FUNCTION_BLOCK TLController (* Composite Function Block Type *)
  (* Standard: 61499-2 *)
  (* Version 0.2, 2003-12-05, JHC, Rockwell Automation, Renamed from NEWCOMPFB. *)
  (* Version 0.1, 2002-01-08, JHC, Rockwell Automation, Added DLY FB as example. *)
  (* Version 0.0, 2000-05-27, JHC, Rockwell Automation *)
  (* Compiler header: package fb.rt.template; *)
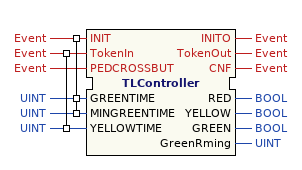
  EVENT_INPUT
    INIT WITH GREENTIME, MINGREENTIME; (* Initialization Request *)
    TokenIn WITH YELLOWTIME;
    PEDCROSSBUT;
  END_EVENT
  EVENT_OUTPUT
    INITO; (* Initialization Confirm *)
    TokenOut;
    CNF;
  END_EVENT
  VAR_INPUT
    GREENTIME : UINT;
    MINGREENTIME : UINT;
    YELLOWTIME : UINT;
  END_VAR
  VAR_OUTPUT
    RED : BOOL;
    YELLOW : BOOL;
    GREEN : BOOL;
    GreenRming : UINT;
  END_VAR
  FBS
    ButPressCTR : E_CTU(PV := 4);
    CLOCK : E_CYCLE(DT := t#1s);
    Split1 : E_SPLIT;
    Controller1 : Controller;
  END_FBS
  EVENT_CONNECTIONS
    PEDCROSSBUT TO ButPressCTR.CU;
    Split1.EO1 TO TokenOut;
    Split1.EO2 TO CLOCK.STOP;
    INIT TO CLOCK.START;
    TokenIn TO CLOCK.START;
    INIT TO Controller1.INIT;
    CLOCK.EO TO Controller1.CLK;
    TokenIn TO Controller1.LD;
    Controller1.INITO TO INITO;
    Controller1.CNF TO CNF;
  END_CONNECTIONS
  DATA_CONNECTIONS
    Controller1.RED TO RED;
    Controller1.YELLOW TO YELLOW;
    Controller1.GREEN TO GREEN;
    Controller1.GREENREMAINING TO GreenRming;
    ButPressCTR.Q TO Controller1.PEDCROSS;
    GREENTIME TO Controller1.GREENTIME;
    MINGREENTIME TO Controller1.MINGREENTIME;
    YELLOWTIME TO Controller1.YELLOWTIME;
  END_CONNECTIONS
END_FUNCTION_BLOCK
